FUNCTION_BLOCK FB_Machine EXTENDS FB_Generic
VAR_INPUT

END_VAR
VAR_OUTPUT

END_VAR
VAR	

	
	stSubModuleInfo		: ARRAY [1..iSubModule] OF ST_PMLSubUnitInfo;	//Informations about the Subunits


	
	
END_VAR
VAR CONSTANT
	iSubModule	: UDINT :=1;
END_VAR

GVL.fb_sample(
	eModeCommand:= eModeCommand, 
	eCommand:= eCommand, 
	eMode=> , 
	eState=> stSubModuleInfo[iSubModule].eState, 
	bUndefinedDone=> , 
	bInvalidModeCommandOut=> , 
	bChangeIntoProduction=> );
stSubModuleInfo[iSubModule].Active		:= TRUE;

IF  GVL.fb_sample.bUndefinedDone  THEN
	bUndefinedDone := TRUE;
END_IF

//The fbStateMachine from FB_Machine gets the Information about the states and activity from the subunits
fbStateMachine.stSubUnitInfoRef.ArraySize		:= SIZEOF(stSubModuleInfo);
fbStateMachine.stSubUnitInfoRef.NoOfSubUnits	:= iSubModule;
fbStateMachine.stSubUnitInfoRef.pArray			:= ADR(stSubModuleInfo);



//Set unit information 
M_SetUnitInfo();


SUPER^();

{attribute 'object_name' := 'M_Clearing'}
METHOD M_Clearing

CASE fbUnitModeManager.eModeStatus OF
	ePMLProtUnitMode_Production:		//Production, Mantainance, Manual
		FOR i:=1 TO MaxAlarms DO
			GVL.pml_adminAlarm.M_AcknowledgeAlarm(stAdmin:=GVL.PackTags.Admin,stAlarm:=GVL.PackTags.Admin.Alarm[i]);
			GVL.pml_adminAlarm.M_ClearAlarm(stAdmin:=GVL.PackTags.Admin,stAlarm:=GVL.PackTags.Admin.Alarm[i]);
		END_FOR			
		IF MAIN.application.safety.M_reset() THEN
			IF MAIN.application.safety.xError THEN
				eCommand	:= ePMLCommand_Abort;
			ELSE
				M_StateComplete();
			END_IF
		END_IF	
		
	
	ePMLProtUnitMode_Maintenance, ePMLProtUnitMode_Manual, ePMLUnitMode_Service:
		M_StateComplete();
END_CASE
END_METHOD

{attribute 'object_name' := 'M_Resetting'}
METHOD M_Resetting
CASE fbUnitModeManager.eModeStatus OF
	ePMLProtUnitMode_Production:		//Production, Mantainance, Manual	
		IF MAIN.application.safety.M_reset() THEN
			IF MAIN.application.safety.xError THEN
				eCommand	:= ePMLCommand_Abort;
			ELSE
				M_StateComplete();
			END_IF
		END_IF	
		
	
	ePMLProtUnitMode_Maintenance, ePMLProtUnitMode_Manual, ePMLUnitMode_Service:
		M_StateComplete();
END_CASE
END_METHOD

METHOD M_SetUnitInfo
VAR_INPUT
END_VAR
GVL.aUnitInfo[eMachine].Name			:= 'fbMachine';
GVL.aUnitInfo[eMachine].ActMode			:= eMode;
GVL.aUnitInfo[eMachine].ActState		:= eState;

GVL.aUnitInfo[eSample].Name				:= 'fb_sample';
GVL.aUnitInfo[eSample].ActMode			:= GVL.fb_sample.eMode;
GVL.aUnitInfo[eSample].ActState			:= GVL.fb_sample.eState;
END_METHOD

{attribute 'object_name' := 'M_Starting'}
METHOD M_Starting
CASE fbUnitModeManager.eModeStatus OF
	ePMLProtUnitMode_Production:		//Production, Mantainance, Manual
		//Resetting all Commands and Value
		G_HMI.bAging_test	:= FALSE;
		M_StateComplete();
	ePMLProtUnitMode_Maintenance, ePMLProtUnitMode_Manual, ePMLUnitMode_Service:
		M_StateComplete();
END_CASE
END_METHOD

END_FUNCTION_BLOCK

(* stored: Version 1.1.0.1, ProductVersion 3.1.4024.12
   POU FB_Machine: Id {8f8b4044-4b54-4b05-9dcb-51655cce136f}, SpecialFunc None
   Method M_Clearing: Id {242a7bec-354c-403a-8360-5cddeab3cb27}
   Method M_Resetting: Id {c82aab94-be7d-4f8e-a811-07458a877516}
   Method M_SetUnitInfo: Id {613978d3-6a85-41f0-ad1f-b7556291b862}
   Method M_Starting: Id {607735ee-5540-4bee-8bb9-efaec3726053} *)
